		ReadStep_MONITOR: // MONITOR
			IF _fbTcpRead.xReady THEN
				IF (_fbTcpRead.udiCount > 0) THEN
					//
					MemSet(
						destAddr:=ADR(strRead),
						fillByte:=0,
						n:=SIZEOF(strRead)); 
					MemSet(
						destAddr:=ADR(byteArrayRead),
						fillByte:=0,
						n:=SIZEOF(byteArrayRead)); 
					MemCpy(
						destAddr:=ADR(strRead),
						srcAddr:=ADR(_ReadData.sString),
						n:=SEL(_fbTcpRead.udiCount > 255, _fbTcpRead.udiCount, 255));
					MemCpy(
						destAddr:=ADR(byteArrayRead),
						srcAddr:=ADR(_ReadData.bArray),
						n:=SEL(_fbTcpRead.udiCount > 255, _fbTcpRead.udiCount, 255));
					MemSet(
						destAddr:=ADR(_ReadData.sString),
						fillByte:=0,
						n:=SIZEOF(_ReadData.sString)); 
					//
					dRecordRead := dRecordRead + 1;
				END_IF
				
			ELSIF _fbTcpRead.xError OR NOT _Read THEN
				_ReadStep := ReadStep_RESET;
				
			END_IF
			 
	END_CASE
	
	bBusyRead := (_ReadStep <> ReadStep_IDLE) AND _fbTcpRead.xBusy;
	_fbTcpRead(xEnable := , 
				itfConnection := _fbTcpClient.itfConnection, 
				udiSize := SIZEOF(_ReadData.bArray), 
				pData := ADR(_ReadData.bArray), 
				udiCount => );

{endregion}

METHOD INTERNAL _M_Reconnect : BOOL
_ConnectStep := ConnectStep_IDLE;
END_METHOD

METHOD INTERNAL _M_Write : BOOL
VAR_INPUT
	Data: STRING(255);
END_VAR
IF bConnected AND NOT bBusyWrite THEN
	bBusyWrite := TRUE; // do this as a workaround to show "busy" ASAP to let callers know to hold back
	_Write:=TRUE;
	_DataToWrite:=Data;
	_M_Write := TRUE;
	
ELSE
	_M_Write := FALSE;
	
END_IF
END_METHOD

END_FUNCTION_BLOCK

// ---- FB/controller/F_DpadState.TcPOU
FUNCTION F_DpadState : ST_Dpad
VAR_INPUT
	State: USINT;
END_VAR

CASE State OF
	0:
		F_DpadState.Up := TRUE;
		F_DpadState.Down := FALSE;
		F_DpadState.Left := FALSE;
		F_DpadState.Right := FALSE;
	1:
		F_DpadState.Up := TRUE;
		F_DpadState.Down := FALSE;
		F_DpadState.Left := FALSE;
		F_DpadState.Right := TRUE;
	2:
		F_DpadState.Up := FALSE;
		F_DpadState.Down := FALSE;
		F_DpadState.Left := FALSE;
		F_DpadState.Right := TRUE;
	3:
		F_DpadState.Up := FALSE;
		F_DpadState.Down := TRUE;
		F_DpadState.Left := FALSE;
		F_DpadState.Right := TRUE;
	4:
		F_DpadState.Up := FALSE;
		F_DpadState.Down := TRUE;
		F_DpadState.Left := FALSE;
		F_DpadState.Right := FALSE;
	5:
		F_DpadState.Up := FALSE;
		F_DpadState.Down := TRUE;
		F_DpadState.Left := TRUE;
		F_DpadState.Right := FALSE;
	6:
		F_DpadState.Up := FALSE;
		F_DpadState.Down := FALSE;
		F_DpadState.Left := TRUE;
		F_DpadState.Right := FALSE;
	7:
		F_DpadState.Up := TRUE;
		F_DpadState.Down := FALSE;
		F_DpadState.Left := TRUE;
		F_DpadState.Right := FALSE;
		
ELSE
	F_DpadState.Up := FALSE;
	F_DpadState.Down := FALSE;
	F_DpadState.Left := FALSE;
	F_DpadState.Right := FALSE;
		
END_CASE

END_FUNCTION

// ---- FB/FB_WriteParameters.TcPOU
FUNCTION_BLOCK FB_WriteParameters
VAR_INPUT
END_VAR
VAR_OUTPUT
END_VAR
VAR
END_VAR

// axis parameters offsets
// https://infosys.beckhoff.com/content/1033/tc3_ads_intro/713091211.html?id=750639462434375559

END_FUNCTION_BLOCK

// ---- FB/F_Checksum.TcPOU
FUNCTION F_Checksum : UINT
VAR_INPUT
	data: POINTER TO BYTE;
	length: UINT;
END_VAR
VAR
	curr_crc: UINT;
	sum1, sum2: USINT;
	_i, _j, _k: UINT;
END_VAR

// https://www.tutorialspoint.com/cyclic-redundancy-check-crc-in-arduino
curr_crc := 16#0000;
sum1 := UINT_TO_USINT(curr_crc);
sum2 := UINT_TO_USINT(SHR(curr_crc, 8));
FOR _i:=0 TO length - 1 BY 1 DO
	sum1 := (sum1 + data[_i]) MOD 255;
	sum2 := (sum2 + sum1) MOD 255;
END_FOR
F_Checksum := SHL(sum2, 8) OR sum1;

END_FUNCTION

// ---- FB/group/FB_RemoveAllAxes.TcPOU
FUNCTION_BLOCK FB_RemoveAllAxes
VAR_INPUT
	Execute				: BOOL;
END_VAR
VAR_IN_OUT
	stGroupRef: AXES_GROUP_REF;
	mcs: ARRAY[1..6] OF AXIS_REF;
END_VAR
VAR_OUTPUT
	Done				: BOOL;
	Busy				: BOOL;
	Error				: BOOL;
END_VAR
VAR
	fbRemoveAxis		: ARRAY[1..6] OF MC_RemoveAxisFromGroup;
	i					: UINT;
END_VAR

Done := TRUE;
Busy := FALSE;
Error := FALSE;

fbRemoveAxis[1].IdentInGroup := MCS_X; //X-Axis
fbRemoveAxis[2].IdentInGroup := MCS_Y; //Y-Axis
fbRemoveAxis[3].IdentInGroup := MCS_Z; //Z-Axis
fbRemoveAxis[4].IdentInGroup := ADDAX1;
fbRemoveAxis[5].IdentInGroup := ADDAX2;
fbRemoveAxis[6].IdentInGroup := ADDAX3;

FOR i:=1 TO 6 DO
	fbRemoveAxis[i](AxesGroup:=stGroupRef, IdentInGroup := mcs[i], Execute := Execute);

	IF (NOT fbRemoveAxis[i].Done) THEN
		Done := FALSE;
	END_IF
	IF (fbRemoveAxis[i].Busy) THEN
		Busy := TRUE;
	END_IF
	IF (fbRemoveAxis[i].Error) THEN
		Error := TRUE;
	END_IF
END_FOR

END_FUNCTION_BLOCK

// ---- FB/jog/F_SetJogButtons.TcPOU
FUNCTION F_SetJogButtons : INT
VAR_INPUT
	CoordinateSystem: SMC_COORD_SYSTEM;
	ABC_as_ACS: BOOL;
END_VAR
VAR
END_VAR

CASE CoordinateSystem OF
	SMC_COORD_SYSTEM.ACS:
		F_SetJogButtons := 0;
	SMC_COORD_SYSTEM.MCS:
		IF ABC_as_ACS THEN
			F_SetJogButtons := 2;
		ELSE
			F_SetJogButtons := 1;
		END_IF
	SMC_COORD_SYSTEM.PCS_1:
		IF ABC_as_ACS THEN
			F_SetJogButtons:= 2;
		ELSE
			F_SetJogButtons := 1;
		END_IF
	SMC_COORD_SYSTEM.PCS_2:
		IF ABC_as_ACS THEN
			F_SetJogButtons := 2;
		ELSE
			F_SetJogButtons := 1;
		END_IF
	SMC_COORD_SYSTEM.TCS:
		IF ABC_as_ACS THEN
			F_SetJogButtons := 2;
		ELSE
			F_SetJogButtons := 1;
		END_IF
	SMC_COORD_SYSTEM.WCS:
		IF ABC_as_ACS THEN
			F_SetJogButtons := 2;
		ELSE
			F_SetJogButtons := 1;
		END_IF
	ELSE
		F_SetJogButtons := 0;
		
END_CASE

END_FUNCTION

// ---- FB/logic/BuildLogicCmd.TcPOU
FUNCTION BuildLogicCmd : STRING(GVL.COMMAND_LEN)
VAR_INPUT
	stCommand: ST_LogicCmd;
END_VAR
VAR
    _Command: STRING(GVL.COMMAND_LEN);
END_VAR
VAR CONSTANT
	_Delimiter: STRING:=' ';
END_VAR

// IF PASS|INPUT|REGISTER|COUNTER <index> >|<|=|>=|<= <value>
// THEN OUTPUT|JUMP|CNTUP|CNTDN|CNTRST|REGISTER|NOP <index> <value>
// ELSE OUTPUT|JUMP|CNTUP|CNTDN|CNTRST|REGISTER|NOP <index> <value>
//
// IF_Condition
// IF_Condition_Idx
// IF_Condition_Operator
// IF_Condition_Operator_Compare
// THEN_Function
// THEN_Function_Value
// THEN_Function_Idx
// ELSE_Function
// ELSE_Function_Idx
// ELSE_Function_Value

// clear the command
_Command:='';

// build command
F_AddElement(_Command, _Delimiter, 'IF');
F_AddElement(_Command, _Delimiter, TO_STRING(stCommand.IF_Condition));
IF stCommand.IF_Condition <> E_LogicIfCondition.PASS THEN
	F_AddElement(_Command, _Delimiter, INT_TO_STRING(stCommand.IF_Condition_Idx));
	F_AddElement(_Command, _Delimiter, TO_STRING(stCommand.IF_Condition_Operator));
	F_AddElement(_Command, _Delimiter, UDINT_TO_STRING(stCommand.IF_Condition_Operator_Value));
END_IF
F_AddElement(_Command, _Delimiter, 'THEN');
F_AddElement(_Command, _Delimiter, TO_STRING(stCommand.THEN_Function));
IF stCommand.THEN_Function <> E_LogicFunction.NOP THEN
	F_AddElement(_Command, _Delimiter, INT_TO_STRING(stCommand.THEN_Function_Idx));
	IF stCommand.THEN_Function = E_LogicFunction.OUTPUT OR 
		stCommand.THEN_Function = E_LogicFunction.REGISTER THEN
			F_AddElement(_Command, _Delimiter, UDINT_TO_STRING(stCommand.THEN_Function_Value));
	END_IF
END_IF
F_AddElement(_Command, _Delimiter, 'ELSE');
F_AddElement(_Command, _Delimiter, TO_STRING(stCommand.ELSE_Function));
IF stCommand.ELSE_Function <> E_LogicFunction.NOP THEN
	F_AddElement(_Command, _Delimiter, INT_TO_STRING(stCommand.ELSE_Function_Idx));
	IF stCommand.ELSE_Function = E_LogicFunction.OUTPUT 
		OR stCommand.ELSE_Function = E_LogicFunction.REGISTER THEN
			F_AddElement(_Command, _Delimiter, UDINT_TO_STRING(stCommand.ELSE_Function_Value));
	END_IF
END_IF

// set function equal to command
BuildLogicCmd := _Command;

END_FUNCTION

// ---- FB/output/BuildOutputCmd.TcPOU
FUNCTION BuildOutputCmd : STRING(GVL.COMMAND_LEN)
VAR_INPUT
	stCommand: ST_OutputCmd;
END_VAR
VAR
    _Command: STRING(GVL.COMMAND_LEN);
END_VAR
VAR CONSTANT
	_Delimiter: STRING:=' ';
	_OutTypeDig: STRING(3):='DIG';
	_OutTypePwm: STRING(3):='PWM';
END_VAR

// DIG +0001.00 +0001.00 (turn digital input 1 on)
// DIG +0001.00 +0000.00 (turn digital input 1 off)
// PWM +0001.00 +0030.00(set PWM 1 to position 30)

// clear the command
_Command:='';

//
CASE stCommand.OutputType OF
	DUT_OutputType.Digital:
		F_AddElement(_Command, _Delimiter, _OutTypeDig);
	DUT_OutputType.Pwm:
		F_AddElement(_Command, _Delimiter, _OutTypePwm);
END_CASE

//
F_AddElement(_Command, _Delimiter, INT_TO_STRING(stCommand.OutputTarget));

//
F_AddElement(_Command, _Delimiter, LREAL_TO_STRING(stCommand.OutputValue1));

// set function equal to command
BuildOutputCmd := _Command;

END_FUNCTION

// ---- FB/pause/BuildPauseCmd.TcPOU
FUNCTION BuildPauseCmd : STRING(GVL.COMMAND_LEN)
VAR_INPUT
	stCommand: ST_PauseCmd;
END_VAR
VAR
    _Command: STRING(GVL.COMMAND_LEN);
END_VAR
VAR CONSTANT
	_Delimiter: STRING:=' ';
END_VAR

// clear the command
_Command:='';

// build command
F_AddElement(_Command, _Delimiter, TIME_TO_STRING(stCommand.PauseTime));

// set function equal to command
BuildPauseCmd := _Command;

END_FUNCTION

// ---- FB/varset/BuildVarSetCmd.TcPOU
FUNCTION BuildVarSetCmd : STRING(GVL.COMMAND_LEN)
VAR_INPUT
	stCommand: ST_VarSetCmd;
END_VAR
VAR
    _Command: STRING(GVL.COMMAND_LEN);
END_VAR
VAR CONSTANT
	_Delimiter: STRING:=' ';
	_ArrayTypeS: STRING(3):='STO';
	_ArrayTypeV: STRING(3):='VIS';
	_ArrayTypeF: STRING(3):='FLG';
END_VAR

// S|V|F index x y z a b c
// S 0000 +0000.00 +0000.00 +0000.00 +0000.00 +0000.00 +0000.00 
// V 0000 +0000.00 +0000.00 +0000.00 +0000.00 +0000.00 +0000.00 
// F 0000 1

// clear the command
_Command:='';

// build the command
CASE stCommand.ArrayType OF
	DUT_Command_ArrayType.StoredPosition:
		F_AddElement(_Command, _Delimiter, _ArrayTypeS);
	DUT_Command_ArrayType.VisionRegister:
		F_AddElement(_Command, _Delimiter, _ArrayTypeV);
	DUT_Command_ArrayType.Flag:
		F_AddElement(_Command, _Delimiter, _ArrayTypeF);
END_CASE

// add the array index
F_AddElement(_Command, _Delimiter, INT_TO_STRING(stCommand.ArrayIndex));

// add the coordinates
IF stCommand.ArrayType = DUT_Command_ArrayType.StoredPosition 
	OR stCommand.ArrayType = DUT_Command_ArrayType.VisionRegister THEN
		F_AddElement(_Command, _Delimiter, LREAL_TO_STRING(stCommand.Coordinates.X));
		F_AddElement(_Command, _Delimiter, LREAL_TO_STRING(stCommand.Coordinates.Y));
		F_AddElement(_Command, _Delimiter, LREAL_TO_STRING(stCommand.Coordinates.Z));
		F_AddElement(_Command, _Delimiter, LREAL_TO_STRING(stCommand.Coordinates.A));
		F_AddElement(_Command, _Delimiter, LREAL_TO_STRING(stCommand.Coordinates.B));
		F_AddElement(_Command, _Delimiter, LREAL_TO_STRING(stCommand.Coordinates.C));
		
ELSIF stCommand.ArrayType = DUT_Command_ArrayType.Flag THEN
		// we only send the x for readability. it will work if we send them all.
		F_AddElement(_Command, _Delimiter, LREAL_TO_STRING(stCommand.Coordinates.X));
		
END_IF

// set function equal to command
BuildVarSetCmd := _Command;

END_FUNCTION

// ---- FB/vision/BuildVisionCmd.TcPOU
FUNCTION BuildVisionCmd : STRING(GVL.COMMAND_LEN)
VAR_INPUT
    stCommand: ST_VisionCmd;
END_VAR
VAR
    _Command: STRING(GVL.COMMAND_LEN);
END_VAR
VAR CONSTANT
	_Delimiter: STRING:=' ';
	_CommandTypeCal: STRING(3):='CAL'; // calibrate vision
	_CommandTypeAcq: STRING(3):='ACQ'; // acquire (capture) image
	_CommandTypeLoc: STRING(3):='LOC'; // locate part
END_VAR

// C|A|L ImageWidth ImageHeight Timeout

// C Calibrate vision system
    // CheckerSize (user units) XCount YCount 
    // C 2016 2000 60 25.0 6 9
    
// A Aquire image
    // A 2016 2000 60
    
// L Locate part 
    // MaxParts MaxOverlap Score ToleranceAngle ResultPostion TemplateName ScriptName
    // L 2016 2000 60 10 0.0 0.8 90.0 1 template.jpg FastTemplateMatching.py
	// MaxParts - max number of parts to find in image
	// MaxOverlap - max overlap of parts in image
	// Score - min required score for parts
	// ToleranceAngle - +/- search angle (the larger the number, the longer the search)
	// ResultPostion - index of vision register to store result
	// TemplateName - name of the template to search for
	// ScriptName - name of the template to search for

// clear the command
_Command:='';

// build the command
CASE stCommand.CommandType OF
	DUT_Command_VisionType.Calibrate:
		F_AddElement(_Command, _Delimiter, _CommandTypeCal);
	DUT_Command_VisionType.Acquire:
		F_AddElement(_Command, _Delimiter, _CommandTypeAcq);
	DUT_Command_VisionType.LocatePart:
		F_AddElement(_Command, _Delimiter, _CommandTypeLoc);
END_CASE

// add the common items width, height, timeout
F_AddElement(_Command, _Delimiter, UINT_TO_STRING(stCommand.ImageWidth));
F_AddElement(_Command, _Delimiter, UINT_TO_STRING(stCommand.ImageHeight));
F_AddElement(_Command, _Delimiter, UDINT_TO_STRING(stCommand.Timeout));

//
CASE stCommand.CommandType OF
	DUT_Command_VisionType.Calibrate:
		// C 2016 2000 60 25.0 6 9
		F_AddElement(_Command, _Delimiter, REAL_TO_STRING(stCommand.Calibrate.CheckerSize));
		F_AddElement(_Command, _Delimiter, UINT_TO_STRING(stCommand.Calibrate.CheckerXCount));
		F_AddElement(_Command, _Delimiter, UINT_TO_STRING(stCommand.Calibrate.CheckerYCount));
		
	DUT_Command_VisionType.Acquire:
		// A 2016 2000 60
		// we are done
		
	DUT_Command_VisionType.LocatePart:
		// L 2016 2000 60 10 0.0 0.8 90.0 1 template.jpg FastTemplateMatching.py
		F_AddElement(_Command, _Delimiter, UINT_TO_STRING(stCommand.Locate.MaxParts));
		F_AddElement(_Command, _Delimiter, REAL_TO_STRING(stCommand.Locate.MaxOverlap));
		F_AddElement(_Command, _Delimiter, REAL_TO_STRING(stCommand.Locate.Score));
		F_AddElement(_Command, _Delimiter, REAL_TO_STRING(stCommand.Locate.ToleranceAngle));
		F_AddElement(_Command, _Delimiter, UINT_TO_STRING(stCommand.Locate.ResultPosition));
		F_AddElement(_Command, _Delimiter, stCommand.Locate.TemplateName);
		F_AddElement(_Command, _Delimiter, stCommand.Locate.ScriptFilename);
		
END_CASE

// set function equal to command
BuildVisionCmd := _Command;

END_FUNCTION

// ---- FB/vision/OpenCV.TcPOU
FUNCTION_BLOCK OpenCV EXTENDS PythonServerHandler

SUPER^();

METHOD PUBLIC M_CalibrateCamera : BOOL
VAR_INPUT
	iImageWidth: UINT:=2016;
	iImageHeight: UINT:=2000;
	uTimeout: UDINT:=60; //sec
	fCalCheckerSize: REAL:=25.0; //mm
	iCalCheckerX: UINT:=6;
	iCalCheckerY: UINT:=9;
END_VAR
VAR
	_Command : STRING(255);
END_VAR
VAR	
	_CalScriptFileName: STRING:='/var/opt/codesys/PlcLogic/Application/Vision/CalibrateCamera.py';
	_CalResultFile: STRING:='/var/opt/codesys/PlcLogic/visu/outputimage.jpg';
END_VAR

// calibrate with a checkerboard
// sudo python /var/opt/codesys/PlcLogic/Application/CalibrateCamera.py -s cal.yaml -l 24.5 -x 6 -y 9 -d false

IF NOT _Busy THEN
	M_CalibrateCamera := TRUE;
	
	_Command := CONCAT('sudo python ', _CalScriptFileName);
	_Command := CONCAT(_Command, ' -l ');
	_Command := CONCAT(_Command, REAL_TO_STRING(fCalCheckerSize));
	_Command := CONCAT(_Command, ' -x ');
	_Command := CONCAT(_Command, UINT_TO_STRING(iCalCheckerX));
	_Command := CONCAT(_Command, ' -y ');
	_Command := CONCAT(_Command, UINT_TO_STRING(iCalCheckerY));
	_Command := CONCAT(_Command, ' -w ');
	_Command := CONCAT(_Command, UINT_TO_STRING(iImageWidth));
	_Command := CONCAT(_Command, ' -h ');
	_Command := CONCAT(_Command, UINT_TO_STRING(iImageHeight));
	_Command := CONCAT(_Command, ' -r ');
	_Command := CONCAT(_Command, _CalResultFile);
	_Command := CONCAT(_Command, ' 2> ./vision_log.txt ');
	
	SUPER^._M_Execute(Command:=_Command, Timeout:=uTimeout);
	
ELSE
	M_CalibrateCamera := FALSE;
	//_Error := TRUE;
	//_ErrorDescription := 'function busy.';
	
END_IF
END_METHOD

METHOD PUBLIC M_CaptureImage : BOOL
VAR_INPUT
	iImageWidth: UINT:=2016;
	iImageHeight: UINT:=2000;
	uTimeout: UDINT:=60; //sec
END_VAR
VAR
	_Command : STRING(255);
END_VAR
VAR
	_ImageScriptFileName: STRING:='/var/opt/codesys/PlcLogic/Application/Vision/CaptureImage.py';
	_CaptureImageName: STRING:='/var/opt/codesys/PlcLogic/visu/outputimage.jpg';
END_VAR

// capture an image
// sudo python /var/opt/codesys/PlcLogic/Application/CaptureImage.py -s /var/opt/codesys/PlcLogic/Application/input.jpg -w 2016 -h 2000

IF NOT _Busy THEN
	M_CaptureImage := TRUE;
	
	_Command := CONCAT('sudo python ', _ImageScriptFileName);
	_Command := CONCAT(_Command, ' -s ');
	_Command := CONCAT(_Command, _CaptureImageName);
	_Command := CONCAT(_Command, ' -w ');
	_Command := CONCAT(_Command, UINT_TO_STRING(iImageWidth));
	_Command := CONCAT(_Command, ' -h ');
	_Command := CONCAT(_Command, UINT_TO_STRING(iImageHeight));
	_Command := CONCAT(_Command, ' 2> ./vision_log.txt ');
	
	SUPER^._M_Execute(Command:=_Command, Timeout:=uTimeout);
	
ELSE
	M_CaptureImage := FALSE;
	//_Error := TRUE;
	//_ErrorDescription := 'function busy.';
	
END_IF
END_METHOD

METHOD PUBLIC M_LocatePart : BOOL
VAR_INPUT
	iImageWidth: UINT:=2016;
	iImageHeight: UINT:=2000;
	uTimeout: UDINT:=60; //sec
	iMaxPos: UINT:=10; // i
	dMaxOverlap: REAL:=0.0; // j
	dScore: REAL:=0.8; // k
	dToleranceAngle: REAL:=90.0; // l
	sTemplateName: STRING:='template.jpg';
	sScriptFilename: STRING:='FastTemplateMatching.py';
END_VAR
VAR
	_Command : STRING(255);
END_VAR
VAR CONSTANT
	//_SCRIPT_FILE_NAME: STRING:='/var/opt/codesys/PlcLogic/Application/Vision/FastTemplateMatching.py';
	_SCRIPT_DIR_PATH: STRING:='/var/opt/codesys/PlcLogic/Application/Vision/';
	_RESULT_FILE_NAME: STRING:='/var/opt/codesys/PlcLogic/visu/outputimage.jpg';
	_TEMPLATE_DIR_PATH: STRING:='/var/opt/codesys/PlcLogic/Application/Vision/Templates/';
END_VAR

// run the designated vision program
// sudo python /var/opt/codesys/PlcLogic/Application/Vision/TemplateMatch.py -s /var/opt/codesys/PlcLogic/visu/outputimage.jpg        -t /var/opt/codesys/PlcLogic/Application/Vision/Template3.JPG -i 0.9 -j 1.0 -d true -w 2016 -h 2000
// sudo python /var/opt/codesys/PlcLogic/Application/Vision/FastTemplateMatching.py -s /var/opt/codesys/PlcLogic/visu/outputimage.jpg -t /var/opt/codesys/PlcLogic/Application/Vision/Template.jpg -w 2016 -h 2000 -d false
IF NOT _Busy THEN
	M_LocatePart := TRUE;
	
	_Command := CONCAT('sudo python ', _SCRIPT_DIR_PATH);
	_Command := CONCAT(_Command, sScriptFilename);
	//_Command := CONCAT(_Command, ' -s '); // need to trim down the string length
	//_Command := CONCAT(_Command, _VisionImageName);
	_Command := CONCAT(_Command, ' -t ');
	_Command := CONCAT(_Command, _TEMPLATE_DIR_PATH);
	_Command := CONCAT(_Command, sTemplateName);
	_Command := CONCAT(_Command, ' -i ');
	_Command := CONCAT(_Command, UINT_TO_STRING(iMaxPos));
	_Command := CONCAT(_Command, ' -j ');
	_Command := CONCAT(_Command, REAL_TO_STRING(dMaxOverlap));
	_Command := CONCAT(_Command, ' -k ');
	_Command := CONCAT(_Command, REAL_TO_STRING(dScore));
	_Command := CONCAT(_Command, ' -l ');
	_Command := CONCAT(_Command, REAL_TO_STRING(dToleranceAngle));
	_Command := CONCAT(_Command, ' -w ');
	_Command := CONCAT(_Command, UINT_TO_STRING(iImageWidth));
	_Command := CONCAT(_Command, ' -h ');
	_Command := CONCAT(_Command, UINT_TO_STRING(iImageHeight));
	_Command := CONCAT(_Command, ' 2> ./vision_log.txt ');
	
	SUPER^._M_Execute(Command:=_Command, Timeout:=uTimeout);
	
ELSE
	M_LocatePart := FALSE;
	//_Error := TRUE;
	//_ErrorDescription := 'function busy.';
	
END_IF
END_METHOD

END_FUNCTION_BLOCK

// ---- FB/vision/ParseVisionCmd.TcPOU
FUNCTION_BLOCK ParseVisionCmd
VAR_INPUT
    Command: STRING(GVL.COMMAND_LEN);
END_VAR
VAR_OUTPUT
    stCommand: ST_VisionCmd;
	Error: BOOL;
	ErrorDescription: STRING;
END_VAR
VAR
	_CmdParams: ARRAY [0..GVL.COMMAND_LEN] OF STRING;
    _CommandType: STRING;
	_StrPosition: INT;
END_VAR
VAR CONSTANT
	_CommandTypeCal: STRING(3):='CAL'; // calibrate vision
	_CommandTypeAcq: STRING(3):='ACQ'; // acquire (capture) image
	_CommandTypeLoc: STRING(3):='LOC'; // locate part
END_VAR

// C|A|L ImageWidth ImageHeight Timeout

// C Calibrate vision system
    // CheckerSize (user units) XCount YCount 
    // C 2016 2000 60 25.0 6 9
    
// A Aquire image
    // A 2016 2000 60
    
// L Locate part 
    // MaxParts MaxOverlap Score ToleranceAngle ResultPostion TemplateName ScriptName
    // L 2016 2000 60 10 0.0 0.8 90.0 1 template.jpg FastTemplateMatching.py
	// MaxParts - max number of parts to find in image
	// MaxOverlap - max overlap of parts in image
	// Score - min required score for parts
	// ToleranceAngle - +/- search angle (the larger the number, the longer the search)
	// ResultPostion - index of vision register to store result
	// TemplateName - name of the template to search for
	// ScriptName - name of the template to search for

Error:=FALSE;
ErrorDescription:='';

// split command string into commands
_CmdParams:=F_SplitCmd(Command:=Command);

_CommandType:= _CmdParams[0];
IF _CommandType = _CommandTypeCal THEN
    // C 2016 2000 0060 025.0 0006 0009
	stCommand.CommandType:=DUT_Command_VisionType.Calibrate;
    stCommand.Calibrate.CheckerSize:=STRING_TO_REAL(_CmdParams[4]);
    stCommand.Calibrate.CheckerXCount:=STRING_TO_UINT(_CmdParams[5]);
    stCommand.Calibrate.CheckerYCount:=STRING_TO_UINT(_CmdParams[6]);
	
	IF stCommand.Calibrate.CheckerSize <= 0
		OR stCommand.Calibrate.CheckerXCount <= 0
		OR stCommand.Calibrate.CheckerYCount <= 0 THEN
			Error:=TRUE;
			ErrorDescription:='Checkerboard configuration incorrect';
			RETURN;
	END_IF
    
ELSIF _CommandType = _CommandTypeAcq THEN
    // A 2016 2000 0060
	stCommand.CommandType:=DUT_Command_VisionType.Acquire;
    
ELSIF _CommandType = _CommandTypeLoc THEN
    // L 2016 2000 0060 0010 000.0 0.8 090.0 001 template.jpg FastTemplatMatching.py
	stCommand.CommandType:=DUT_Command_VisionType.LocatePart;
    stCommand.Locate.MaxParts:=STRING_TO_UINT(_CmdParams[4]);
    stCommand.Locate.MaxOverlap:=STRING_TO_REAL(_CmdParams[5]);
    stCommand.Locate.Score:=STRING_TO_REAL(_CmdParams[6]);
    stCommand.Locate.ToleranceAngle:=STRING_TO_REAL(_CmdParams[7]);
    stCommand.Locate.ResultPosition:=STRING_TO_UINT(_CmdParams[8]);
    stCommand.Locate.TemplateName:=_CmdParams[9];
    stCommand.Locate.ScriptFilename:=_CmdParams[10];
	
	IF stCommand.Locate.MaxParts <= 0
		OR stCommand.Locate.ResultPosition < GVL.VIS_ARR_BEG
		OR stCommand.Locate.ResultPosition > GVL.VIS_ARR_END
		OR stCommand.Locate.TemplateName = '' THEN
			Error:=TRUE;
			ErrorDescription:='Locate part configuration incorrect';
			RETURN;
	END_IF
	
ELSE
	Error:=TRUE;
	ErrorDescription:='Unknown command type for vision';
	RETURN;
    
END_IF

// common
stCommand.ImageWidth:=STRING_TO_UINT(_CmdParams[1]);
stCommand.ImageHeight:=STRING_TO_UINT(_CmdParams[2]);
stCommand.Timeout:=STRING_TO_UDINT(_CmdParams[3]);

IF stCommand.ImageWidth <= 0
	OR stCommand.ImageHeight <= 0 THEN
		Error:=TRUE;
		ErrorDescription:='Image size settings incorrect';
END_IF

END_FUNCTION_BLOCK

// ---- FB/vision/VisionCmdProcessor.TcPOU
FUNCTION_BLOCK VisionCmdProcessor EXTENDS Module
VAR_INPUT
	Command: STRING(GVL.COMMAND_LEN):='';
	LogicCmdIO: REFERENCE TO ST_LogicCmdIO;
	VisionSystemIpAddress: STRING(19):='127.0.0.1';
	VisionSystemPort: UINT:=50011;
END_VAR
VAR_OUTPUT
	VisionStateText: STRING:='READY';
END_VAR
VAR
	_CaptureImage_Output: STRING(255);
	_CaptureImage_WorkerUid: STRING;
	_LocatePart_Output: STRING(255);
	_LocatePart_WorkerUid: STRING;
	_RunCalibration_Output: STRING(255);
	_RunCalibration_WorkerUid: STRING;
    _Vision: OpenCV;
    _VisionCommandParser: ParseVisionCmd;
    _VisionDoneRtrig: R_TRIG;
	_VisionBusyRtrig: R_TRIG;
	_VisionResult: STRING(255);
	_ResultPosition: INT;
	_ResultPosition_CAL: INT;
	_ResultPosition_LOC: INT;
	_ResultPosition_CAP: INT;
	_SpacePosition: INT;
	_VisionObjectIndex: UINT;
	_VisionRatio: REAL;
	_VisionRotation: REAL;
	_VisionError: REAL;
	_PartsCount: UDINT;
	_UnitModeCurrentState: PACK_ML.State;
END_VAR

VAR CONSTANT
	_RESPONSE_CAL:          STRING:='res: CAL ';
	_RESPONSE_LOC:          STRING:='res: LOC ';
	_RESPONSE_CAP:          STRING:='res: CAP ';

	_STEP_DONE: 			INT := 1000;
	_STEP_IDLE: 			INT := 0000;
	_STEP_COMMAND: 			INT := 0020;
	_STEP_TRIGGER: 			INT := 0030;
	_STEP_WAIT: 			INT := 0040;
	_STEP_ERR: 				INT := 0050;
END_VAR

SUPER^();

// PackML state machine implementation
_UnitModeCurrentState := SUPER^._UnitMode.CurrentState;

//
CASE SUPER^._SeqMain OF
	
    _STEP_DONE:
		SUPER^._SeqMain := _STEP_IDLE;
        
    _STEP_IDLE:
		// hang out here until called to run
        
    _STEP_COMMAND: // parse vision command
        _VisionCommandParser(Command:=Command);
		IF _VisionCommandParser.Error THEN
			SUPER^.M_Error(Description:=_VisionCommandParser.ErrorDescription);
			//
			SUPER^._SeqMain := _STEP_ERR;
		ELSE
			IF _VisionCommandParser.stCommand.Timeout > 0 THEN
				SUPER^._TimeoutTimer.PT := UDINT_TO_TIME(_VisionCommandParser.stCommand.Timeout * 1000);
			END_IF
			//
			SUPER^._SeqMain := _STEP_TRIGGER;
		END_IF
		
	_STEP_TRIGGER: //
		CASE _VisionCommandParser.stCommand.CommandType OF
			DUT_Command_VisionType.Calibrate: //
				_Vision.M_CalibrateCamera(	iImageWidth:= _VisionCommandParser.stCommand.ImageWidth, 
											iImageHeight:= _VisionCommandParser.stCommand.ImageHeight, 
											fCalCheckerSize:= _VisionCommandParser.stCommand.Calibrate.CheckerSize, 
											iCalCheckerX:= _VisionCommandParser.stCommand.Calibrate.CheckerXCount, 
											iCalCheckerY:= _VisionCommandParser.stCommand.Calibrate.CheckerYCount,
                                            uTimeout:=_VisionCommandParser.stCommand.Timeout);
			
			DUT_Command_VisionType.Acquire: //
				_Vision.M_CaptureImage(	iImageWidth:= _VisionCommandParser.stCommand.ImageWidth, 
										iImageHeight:= _VisionCommandParser.stCommand.ImageHeight,
                                        uTimeout:=_VisionCommandParser.stCommand.Timeout);
			
			DUT_Command_VisionType.LocatePart: //
				_PartsCount := 0;
				LogicCmdIO.Register[_VisionCommandParser.stCommand.Locate.ResultPosition] := 0;
				_Vision.M_LocatePart( 	iImageWidth:= _VisionCommandParser.stCommand.ImageWidth, 
										iImageHeight:= _VisionCommandParser.stCommand.ImageHeight, 
										iMaxPos:= _VisionCommandParser.stCommand.Locate.MaxParts, 
										dMaxOverlap:= _VisionCommandParser.stCommand.Locate.MaxOverlap, 
										dScore:= _VisionCommandParser.stCommand.Locate.Score, 
										dToleranceAngle:= _VisionCommandParser.stCommand.Locate.ToleranceAngle,
                                        uTimeout:=_VisionCommandParser.stCommand.Timeout,
										sTemplateName:=_VisionCommandParser.stCommand.Locate.TemplateName,
										sScriptFilename:=_VisionCommandParser.stCommand.Locate.ScriptFilename);
			
		END_CASE;
		
		//
		SUPER^._SeqMain := _STEP_WAIT;
		
	_STEP_WAIT: //
		IF _VisionDoneRtrig.Q THEN
			
			//
			_VisionResult := _Vision.P_Response;
			
			//
			_ResultPosition_CAL := FIND(STR1:=_VisionResult,STR2:=_RESPONSE_CAL);
			_ResultPosition_LOC := FIND(STR1:=_VisionResult,STR2:=_RESPONSE_LOC);
			_ResultPosition_CAP := FIND(STR1:=_VisionResult,STR2:=_RESPONSE_CAP);
			
			//
			IF _ResultPosition_CAL > 0 THEN 
				// calibration was completed
				// res: CAL rat:23.23 rot:23.23 err:23.23
				_VisionResult := MID(STR:=_VisionResult,LEN:=LEN(_VisionResult)-LEN(_RESPONSE_CAL),POS:=LEN(_RESPONSE_CAL)+1);
				//VisionStateText := CONCAT(VisionStateText, '\n');
				//VisionStateText := CONCAT(VisionStateText, _VisionResult);
				// rat:23.23 rot:23.23 err:23.23
				_ResultPosition := FIND(STR1:=_VisionResult,STR2:='rat:');
				IF _ResultPosition > 0 THEN
					_VisionResult := MID(STR:=_VisionResult,LEN:=LEN(_VisionResult)-LEN('rat:'),POS:=LEN('rat:')+1);
					_SpacePosition := FIND(STR1:=_VisionResult,STR2:=' ');
					_VisionRatio := STRING_TO_REAL(MID(STR:=_VisionResult,LEN:=_SpacePosition-1,POS:=1));
					_VisionResult := MID(STR:=_VisionResult,LEN:=LEN(_VisionResult)-_SpacePosition,POS:=_SpacePosition+1);
				END_IF
				// rot:23.23 err:23.23
				_ResultPosition := FIND(STR1:=_VisionResult,STR2:='rot:');
				IF _ResultPosition > 0 THEN
					_VisionResult := MID(STR:=_VisionResult,LEN:=LEN(_VisionResult)-LEN('rot:'),POS:=LEN('rot:')+1);
					_SpacePosition := FIND(STR1:=_VisionResult,STR2:=' ');
					_VisionRotation := STRING_TO_REAL(MID(STR:=_VisionResult,LEN:=_SpacePosition-1,POS:=1));
					_VisionResult := MID(STR:=_VisionResult,LEN:=LEN(_VisionResult)-_SpacePosition,POS:=_SpacePosition+1);
				END_IF
				// err:23.23
				_ResultPosition := FIND(STR1:=_VisionResult,STR2:='err:');
				IF _ResultPosition > 0 THEN
					_VisionResult := MID(STR:=_VisionResult,LEN:=LEN(_VisionResult)-LEN('err:'),POS:=LEN('err:')+1);
					_SpacePosition := FIND(STR1:=_VisionResult,STR2:=' ');
					_VisionError := STRING_TO_REAL(MID(STR:=_VisionResult,LEN:=_SpacePosition-1,POS:=1));
					_VisionResult := MID(STR:=_VisionResult,LEN:=LEN(_VisionResult)-_SpacePosition,POS:=_SpacePosition+1);
				END_IF
				
			ELSIF _ResultPosition_LOC > 0 THEN 
				// part was located
				// 'res: LOC obj:0 cx:54.66 cy:119.45 a:-12.87 s:0.84 $NLOC obj:1 cx:71.49 cy:100.06 a:10.13 s:0.83 $N'
				_VisionResult := MID(STR:=_VisionResult,LEN:=LEN(_VisionResult)-LEN(_RESPONSE_LOC),POS:=LEN(_RESPONSE_LOC)+1);
				//VisionStateText := CONCAT(VisionStateText, '\n');
				//VisionStateText := CONCAT(VisionStateText, _VisionResult);
				_VisionObjectIndex := 0;
				WHILE FIND(STR1:=_VisionResult,STR2:='obj:') > 0 
					AND _VisionObjectIndex <= _VisionCommandParser.stCommand.Locate.MaxParts 
					AND _VisionObjectIndex + _VisionCommandParser.stCommand.Locate.ResultPosition < GVL.VIS_ARR_END DO
					// 'obj:0 cx:54.66 cy:119.45 a:-12.87 s:0.84 $NLOC obj:1 cx:71.49 cy:100.06 a:10.13 s:0.83 $N'
					// $NLOC obj:1 cx:71.49 cy:100.06 a:10.13 s:0.83 $N'
					_ResultPosition := FIND(STR1:=_VisionResult,STR2:='obj:');
					IF _ResultPosition > 0 THEN
						_PartsCount := _PartsCount + 1;
						_VisionResult := MID(STR:=_VisionResult,LEN:=LEN(_VisionResult)-_ResultPosition-LEN('obj:')+1,POS:=_ResultPosition+LEN('obj:'));
						_SpacePosition := FIND(STR1:=_VisionResult,STR2:=' ');
						_VisionObjectIndex := STRING_TO_UINT(MID(STR:=_VisionResult,LEN:=_SpacePosition-1,POS:=1));
						SUPER^.VisionRegisters[_VisionCommandParser.stCommand.Locate.ResultPosition + _VisionObjectIndex].Comment := CONCAT('obj:', UDINT_TO_STRING(_VisionObjectIndex));
						_VisionResult := MID(STR:=_VisionResult,LEN:=LEN(_VisionResult)-_SpacePosition,POS:=_SpacePosition+1);
					END_IF
					// cx:54.66 cy:119.45 a:-12.87 s:0.84 $NLOC obj:1 cx:71.49 cy:100.06 a:10.13 s:0.83 $N'
					_ResultPosition := FIND(STR1:=_VisionResult,STR2:='cx:');
					IF _ResultPosition > 0 THEN
						_VisionResult := MID(STR:=_VisionResult,LEN:=LEN(_VisionResult)-LEN('cx:'),POS:=LEN('cx:')+1);
						_SpacePosition := FIND(STR1:=_VisionResult,STR2:=' ');
						SUPER^.VisionRegisters[_VisionCommandParser.stCommand.Locate.ResultPosition + _VisionObjectIndex].Position.X := STRING_TO_LREAL(MID(STR:=_VisionResult,LEN:=_SpacePosition-1,POS:=1));
						_VisionResult := MID(STR:=_VisionResult,LEN:=LEN(_VisionResult)-_SpacePosition,POS:=_SpacePosition+1);
					END_IF
					// cy:119.45 a:-12.87 s:0.84 $NLOC obj:1 cx:71.49 cy:100.06 a:10.13 s:0.83 $N'
					_ResultPosition := FIND(STR1:=_VisionResult,STR2:='cy:');
					IF _ResultPosition > 0 THEN
						_VisionResult := MID(STR:=_VisionResult,LEN:=LEN(_VisionResult)-LEN('cy:'),POS:=LEN('cy:')+1);
						_SpacePosition := FIND(STR1:=_VisionResult,STR2:=' ');
						SUPER^.VisionRegisters[_VisionCommandParser.stCommand.Locate.ResultPosition + _VisionObjectIndex].Position.Y := STRING_TO_LREAL(MID(STR:=_VisionResult,LEN:=_SpacePosition-1,POS:=1));
						_VisionResult := MID(STR:=_VisionResult,LEN:=LEN(_VisionResult)-_SpacePosition,POS:=_SpacePosition+1);
					END_IF
					// a:-12.87 s:0.84 $NLOC obj:1 cx:71.49 cy:100.06 a:10.13 s:0.83 $N'
					_ResultPosition := FIND(STR1:=_VisionResult,STR2:='a:');
					IF _ResultPosition > 0 THEN
						_VisionResult := MID(STR:=_VisionResult,LEN:=LEN(_VisionResult)-LEN('a:'),POS:=LEN('a:')+1);
						_SpacePosition := FIND(STR1:=_VisionResult,STR2:=' ');
						SUPER^.VisionRegisters[_VisionCommandParser.stCommand.Locate.ResultPosition + _VisionObjectIndex].Position.A := STRING_TO_LREAL(MID(STR:=_VisionResult,LEN:=_SpacePosition-1,POS:=1));
						_VisionResult := MID(STR:=_VisionResult,LEN:=LEN(_VisionResult)-_SpacePosition,POS:=_SpacePosition+1);
					END_IF
					// s:0.84 $NLOC obj:1 cx:71.49 cy:100.06 a:10.13 s:0.83 $N'
					_ResultPosition := FIND(STR1:=_VisionResult,STR2:='s:');
					IF _ResultPosition > 0 THEN
						_VisionResult := MID(STR:=_VisionResult,LEN:=LEN(_VisionResult)-LEN('s:'),POS:=LEN('s:')+1);
						_SpacePosition := FIND(STR1:=_VisionResult,STR2:=' ');
						SUPER^.VisionRegisters[_VisionCommandParser.stCommand.Locate.ResultPosition + _VisionObjectIndex].Scaling := STRING_TO_REAL(MID(STR:=_VisionResult,LEN:=_SpacePosition-1,POS:=1));
						_VisionResult := MID(STR:=_VisionResult,LEN:=LEN(_VisionResult)-_SpacePosition,POS:=_SpacePosition+1);
					END_IF
					// $NLOC obj:1 cx:71.49 cy:100.06 a:10.13 s:0.83 $N'
				END_WHILE
				// return how many part were found
				LogicCmdIO.Register[_VisionCommandParser.stCommand.Locate.ResultPosition] := _PartsCount;
				
			ELSIF _ResultPosition_CAP > 0 THEN 
				// image was captured
				
			END_IF
			
			//
			SUPER^._SeqMain := _STEP_DONE;
			
		END_IF

END_CASE

//
_Vision(sIpAddress:= VisionSystemIpAddress, uPort:= VisionSystemPort);

//
_VisionBusyRtrig(clk:=_Vision.P_Busy);
IF _VisionBusyRtrig.Q THEN
	VisionStateText := 'BUSY';
END_IF

//
_VisionDoneRtrig(clk:=_Vision.P_Done);
IF _VisionDoneRtrig.Q THEN
	VisionStateText := 'DONE.';
	VisionStateText := CONCAT(VisionStateText, ' Found ');
	VisionStateText := CONCAT(VisionStateText, UDINT_TO_STRING(_PartsCount));
	VisionStateText := CONCAT(VisionStateText, ' parts.');
END_IF

METHOD PROTECTED M_Aborting : BOOL
CASE _SeqAborting OF
	0:
		_Vision.M_Cancel();
		_SeqAborting := _SeqAborting + 1;
		
	1: 
		IF NOT _Vision.P_Busy THEN
			SUPER^.M_StateComplete();
			_SeqAborting := 0;
		END_IF
END_CASE
END_METHOD

METHOD PROTECTED M_Complete : BOOL
// once complete, reset to get back to idle
SUPER^._UnitMode.Reset();
END_METHOD

METHOD PROTECTED M_Execute : BOOL
// here we want to execute our commands/jobs/etc and set completed when done.
IF SUPER^._SeqMain =_STEP_IDLE THEN
	SUPER^.M_StateComplete();
END_IF
END_METHOD

METHOD M_ReconnectVisionSystem : BOOL
// TODO may want to make sure the state machine is not in execute?
_Vision.M_Reconnect();
END_METHOD

METHOD PROTECTED M_Resetting : BOOL
CASE SUPER^._SeqResetting OF
	0:
		_Vision.M_Reset();
		_SeqResetting := _SeqResetting + 1;
	1:
		IF NOT _Vision.P_Error THEN
			//VisionStateText := 'RESET';
			SUPER^.M_StateComplete();
			_SeqResetting := 0;
		END_IF
END_CASE
END_METHOD

METHOD PROTECTED M_SetPackML : BOOL
SUPER^._UnitMode(	sName := 'Vision Processor',
				eInitialState := PACK_ML.State.Idle,
				xActive := TRUE);
END_METHOD

METHOD PROTECTED M_Starting : BOOL
// here we want to clear things and get ready for the execute state
// I can consider this the "INIT" state
SUPER^._SeqMain := _STEP_COMMAND;
SUPER^.M_StateComplete();
END_METHOD

{attribute 'monitoring' := 'variable'}
PROPERTY P_PartsCount : REFERENCE TO UDINT
GET
P_PartsCount REF= _PartsCount;
END_GET
END_PROPERTY

{attribute 'monitoring' := 'variable'}
PROPERTY P_VisionSystemConnected : REFERENCE TO BOOL
GET
P_VisionSystemConnected REF= _Vision._TcpClient.bConnected;
END_GET
END_PROPERTY

END_FUNCTION_BLOCK

// ---- POUs/_10_HMI.TcPOU
PROGRAM _10_HMI
VAR	
	
	SelectedProgramNumber: INT;
	SelectedRecipeRowIndex: INT;
	RecipeRowSelected: BOOL;
	InsertLineAbove: BOOL;
	InsertLineBelow: BOOL;
	DeleteLine: BOOL;
	CopySelectedCommand: BOOL;
	CopiedCommandType: DUT_CommandType;
	CopiedCommandString: STRING(GVL.COMMAND_LEN);
	CopiedCommandComment: STRING;
	PasteCommand: BOOL;
	
	_i,_j,_k: INT;
	
	SetStoredPositionAsCurrent: BOOL;
	SelectedStoredPosition: UINT;
	SetVisionRegisterAsCurrent: BOOL;
	SelectedVisionRegister: UINT;
	SelectedFlag: UINT;
	
	//
	TeachPosition: BOOL;
	stTeachPosition: ST_MoveCmd;
	
	//
	MoveCmdParser: ParseMoveCmd;
	stMoveCmd: ST_MoveCmd;
	MoveCmdVisu: AddMoveCmd_VISU_STRUCT;
	
	//
	OutputCmdParser: ParseOutputCmd;
	stOutputCmd: ST_OutputCmd;
	OutputCmdVisu: AddOutputCmd_VISU_STRUCT;
	
	//
	PauseCmdParser: ParsePauseCmd;
	stPauseCmd: ST_PauseCmd;
	PauseCmdVisu: AddPauseCmd_VISU_STRUCT;
	
	//
	VisionCmdParser : ParseVisionCmd;
	stVisionCmd : ST_VisionCmd;
	VisionCmdVisu: AddVisionCmd_VISU_STRUCT;
	
	//
	VarSetCmdParser : ParseVarSetCmd;
	stVarSetCmd : ST_VarSetCmd;
	VarSetCmdVisu: AddVarSetCmd_VISU_STRUCT;
	
	//
	LogicCmdParser : ParseLogicCmd;
	stLogicCmd : ST_LogicCmd;
	LogicCmdVisu: AddLogicCmd_VISU_STRUCT;
	
	//
	CurrentVisu: STRING;
	OpenDialog: VU.FbOpenDialogExtended;
    
    // vision
   	HostName   : STRING;
	VisionSystemUrl: STRING;
	VisionOutputImageUrl: STRING;
	VisionSystemIpAddress_Last: STRING(19);

END_VAR

VAR CONSTANT
	LocalIpAddress: STRING(19):='127.0.0.1';
END_VAR

//
IF GVL.StorePersist THEN
	GVL.StorePersist := FALSE;
	// TODO manually store persistent data here.
	// not currently a straight forward way of doing this.
END_IF

//
IF (InsertLineAbove OR InsertLineBelow) AND RecipeRowSelected THEN
	//
	IF InsertLineAbove THEN
		InsertLineAbove := FALSE;
		_j := SelectedRecipeRowIndex + 1;
	ELSIF InsertLineBelow THEN
		InsertLineBelow := FALSE;
		_j := SelectedRecipeRowIndex + 2;
	END_IF
	//
	FOR _i := GVL.PROG_CMDS_ARR_END TO _j BY -1 DO
		// shift all data
		IF _i >= GVL.PROG_CMDS_ARR_BEG AND _i <= GVL.PROG_CMDS_ARR_END THEN // can never really bo too careful am I right?
			PersistentVars.Programs[SelectedProgramNumber].Commands[_i].CommandType := PersistentVars.Programs[SelectedProgramNumber].Commands[_i - 1].CommandType;
			PersistentVars.Programs[SelectedProgramNumber].Commands[_i].CommandString := PersistentVars.Programs[SelectedProgramNumber].Commands[_i - 1].CommandString;
			PersistentVars.Programs[SelectedProgramNumber].Commands[_i].CommandComment := PersistentVars.Programs[SelectedProgramNumber].Commands[_i - 1].CommandComment;
		END_IF
	END_FOR
	//
	PersistentVars.Programs[SelectedProgramNumber].Commands[_j - 1].CommandType := DUT_CommandType.Disabled;
	PersistentVars.Programs[SelectedProgramNumber].Commands[_j - 1].CommandString := '';
	PersistentVars.Programs[SelectedProgramNumber].Commands[_j - 1].CommandComment := '';
END_IF

//
IF DeleteLine AND RecipeRowSelected THEN
	DeleteLine := FALSE;
	FOR _i := SelectedRecipeRowIndex TO GVL.PROG_CMDS_ARR_END - 1 BY 1 DO
		IF _i >= GVL.PROG_CMDS_ARR_BEG AND _i <= GVL.PROG_CMDS_ARR_END THEN // can never really bo too careful am I right?
			PersistentVars.Programs[SelectedProgramNumber].Commands[_i].CommandType := PersistentVars.Programs[SelectedProgramNumber].Commands[_i + 1].CommandType;
			PersistentVars.Programs[SelectedProgramNumber].Commands[_i].CommandString := PersistentVars.Programs[SelectedProgramNumber].Commands[_i + 1].CommandString;
			PersistentVars.Programs[SelectedProgramNumber].Commands[_i].CommandComment := PersistentVars.Programs[SelectedProgramNumber].Commands[_i + 1].CommandComment;
		END_IF
	END_FOR
END_IF

//
IF SetStoredPositionAsCurrent THEN
	SetStoredPositionAsCurrent := FALSE;
	PersistentVars.StoredPositions[SelectedStoredPosition].Position.X := F_RoundLreal(_00_Main.ProcessJog.Position.v[0],2);
	PersistentVars.StoredPositions[SelectedStoredPosition].Position.Y := F_RoundLreal(_00_Main.ProcessJog.Position.v[1],2);
	PersistentVars.StoredPositions[SelectedStoredPosition].Position.Z := F_RoundLreal(_00_Main.ProcessJog.Position.v[2],2);
	PersistentVars.StoredPositions[SelectedStoredPosition].Position.A := F_RoundLreal(_00_Main.ProcessJog.Position.v[3],2);
	PersistentVars.StoredPositions[SelectedStoredPosition].Position.B := F_RoundLreal(_00_Main.ProcessJog.Position.v[4],2);
	PersistentVars.StoredPositions[SelectedStoredPosition].Position.C := F_RoundLreal(_00_Main.ProcessJog.Position.v[5],2);
END_IF

//
IF TeachPosition THEN
	TeachPosition := FALSE;
	//
	stTeachPosition.MoveType := DUT_Command_MoveType.DirectMove;
	stTeachPosition.Speed := 50;
	stTeachPosition.PositionType := DUT_Command_PositionType.AbsolutePosition;
	stTeachPosition.CoordSystem := _00_Main.ProcessJog.CoordSystem;
	stTeachPosition.CoordRef.X := F_RoundLreal(_00_Main.ProcessJog.Position.v[0],2);
	stTeachPosition.CoordRef.Y := F_RoundLreal(_00_Main.ProcessJog.Position.v[1],2);
	stTeachPosition.CoordRef.Z := F_RoundLreal(_00_Main.ProcessJog.Position.v[2],2);
	stTeachPosition.CoordRef.A := F_RoundLreal(_00_Main.ProcessJog.Position.v[3],2);
	stTeachPosition.CoordRef.B := F_RoundLreal(_00_Main.ProcessJog.Position.v[4],2);
	stTeachPosition.CoordRef.C := F_RoundLreal(_00_Main.ProcessJog.Position.v[5],2);
	PersistentVars.Programs[SelectedProgramNumber].Commands[SelectedRecipeRowIndex].CommandType := DUT_CommandType.MoveCommand;
	PersistentVars.Programs[SelectedProgramNumber].Commands[SelectedRecipeRowIndex].CommandString := BuildMoveCmd(stTeachPosition);
	PersistentVars.Programs[SelectedProgramNumber].Commands[SelectedRecipeRowIndex].CommandComment := 'Taught position';
END_IF

//
IF PasteCommand THEN
	PasteCommand := FALSE;
	PersistentVars.Programs[SelectedProgramNumber].Commands[SelectedRecipeRowIndex].CommandType := CopiedCommandType;
	PersistentVars.Programs[SelectedProgramNumber].Commands[SelectedRecipeRowIndex].CommandString := CopiedCommandString;
	PersistentVars.Programs[SelectedProgramNumber].Commands[SelectedRecipeRowIndex].CommandComment := CopiedCommandComment;
END_IF

//
IF CopySelectedCommand THEN
	CopySelectedCommand := FALSE;
	
	//
	CopiedCommandType := PersistentVars.Programs[SelectedProgramNumber].Commands[SelectedRecipeRowIndex].CommandType;
	CopiedCommandString := PersistentVars.Programs[SelectedProgramNumber].Commands[SelectedRecipeRowIndex].CommandString;
	CopiedCommandComment := PersistentVars.Programs[SelectedProgramNumber].Commands[SelectedRecipeRowIndex].CommandComment;
	
	CASE PersistentVars.Programs[SelectedProgramNumber].Commands[SelectedRecipeRowIndex].CommandType OF
		DUT_CommandType.Disabled:
			//
			
		DUT_CommandType.MoveCommand:
			MoveCmdParser(Command := PersistentVars.Programs[SelectedProgramNumber].Commands[SelectedRecipeRowIndex].CommandString);
			stMoveCmd := MoveCmdParser.stCommand;
			
		DUT_CommandType.PauseCommand:
			PauseCmdParser(Command:=PersistentVars.Programs[SelectedProgramNumber].Commands[SelectedRecipeRowIndex].CommandString);
			stPauseCmd := PauseCmdParser.stCommand;
			
		DUT_CommandType.InputCommand:
			//
			
		DUT_CommandType.OutputCommand:
			OutputCmdParser(Command:=PersistentVars.Programs[SelectedProgramNumber].Commands[SelectedRecipeRowIndex].CommandString);
			stOutputCmd := OutputCmdParser.stCommand;
			
		DUT_CommandType.VisionCommand:
			VisionCmdParser(Command:=PersistentVars.Programs[SelectedProgramNumber].Commands[SelectedRecipeRowIndex].CommandString);
			stVisionCmd := VisionCmdParser.stCommand;
			
		DUT_CommandType.VarSetCommand:
			VarSetCmdParser(Command:=PersistentVars.Programs[SelectedProgramNumber].Commands[SelectedRecipeRowIndex].CommandString);
			stVarSetCmd := VarSetCmdParser.stCommand;
			
		DUT_CommandType.CncCommand:
			CncCmdParser(Command:=PersistentVars.Programs[SelectedProgramNumber].Commands[SelectedRecipeRowIndex].CommandString);
			stCncCmd := CncCmdParser.stCommand;
			
		DUT_CommandType.LogicCommand:
			LogicCmdParser(Command:=PersistentVars.Programs[SelectedProgramNumber].Commands[SelectedRecipeRowIndex].CommandString);
			stLogicCmd := LogicCmdParser.stCommand;
			
	END_CASE
	
END_IF

// should be called after CopySelectedCommand case statement
CurrentVisu := VisuElems.CurrentVisu;
OpenDialog(
	xExecute:= , 
	xDone=> , 
	xBusy=> , 
	xError=> , 
	itfClientFilter:= , 
	eError=> , 
	sDialogName:= , 
	xModal:= TRUE, // TRUE - visu in background cannot be used
	pTopLeftPosition:= , 
	itfDialogOpenedListener:= , 
	pbyDialogInterfaceData:= , 
	udiDialogInterfaceDataSize:= , 
	itfDialogCloseListener:= , 
	pbyTagForDialogClosed:= , 
	dwDialogFlags:= );
IF (OpenDialog.xExecute AND OpenDialog.xDone) 
	OR OpenDialog.xError 
	THEN
		OpenDialog.xExecute := FALSE;
END_IF

// used to show the output image on the visu
// 'http://ArfBot:5000/output'
IF  PersistentVars.VisionSystemIpAddress <> VisionSystemIpAddress_Last THEN
	 VisionSystemIpAddress_Last :=  PersistentVars.VisionSystemIpAddress;
	//
	IF PersistentVars.VisionSystemIpAddress = LocalIpAddress THEN
		// https://forge.codesys.com/forge/talk/Runtime/thread/61d60a9fb7/
		SysSockGetHostName(szHostName:=HostName, diNameLen:=SIZEOF(HostName));
		VisionSystemUrl := CONCAT('http://', HostName);
	ELSE
		VisionSystemUrl := CONCAT('http://', PersistentVars.VisionSystemIpAddress);
	END_IF
	//
	VisionSystemUrl := CONCAT(VisionSystemUrl, ':5000');
	VisionOutputImageUrl := CONCAT(VisionSystemUrl,'/output');
END_IF

END_PROGRAM

// ---- DUTs/CommandType.TcTLO
TEXTLIST CommandType
  0 = 'DISABLE'
  1 = 'MOVE'
  2 = 'PAUSE'
  3 = 'INPUT'
  4 = 'OUTPUT'
  5 = 'VISION'
  6 = 'CNC'
  7 = 'VARSET'
  8 = 'LOGIC'
   = ''
END_TEXTLIST

// ---- FB/move/CircleMode.TcTLO
TEXTLIST CircleMode
  0 = 'Border'
  1 = 'Center'
  2 = 'Radius'
   = ''
END_TEXTLIST

// ---- FB/move/CoordSystem.TcTLO
TEXTLIST CoordSystem
  0 = 'ACS'
  1 = 'MCS'
  2 = 'WCS'
  3 = 'PCS_1'
  4 = 'PCS_2'
  5 = 'TCS'
  6 = 'ICS'
   = ''
END_TEXTLIST

// ---- FB/move/MoveType.TcTLO
TEXTLIST MoveType
  0 = 'Circular'
  1 = 'Direct'
  2 = 'Linear'
   = ''
END_TEXTLIST

// ---- FB/move/PathChoice.TcTLO
TEXTLIST PathChoice
  0 = 'Clockwise'
  1 = 'CounterClockwise'
   = ''
END_TEXTLIST

// ---- FB/move/PositionType.TcTLO
TEXTLIST PositionType
  0 = 'Absolute'
  1 = 'Relative'
   = ''
END_TEXTLIST

// ---- FB/output/OutputType.TcTLO
TEXTLIST OutputType
  0 = 'Digital'
  1 = 'PWM'
   = ''
END_TEXTLIST
